// TIA Portal project "PID 2" (V17)

(* hardware
DEVICE "S7-1500/ET200MP station_1"  S7-1500 station
   slot 0: "Rail_0"  Rack  6ES7 590-1***0-0AA0
   slot 1: "PLC_1"  CPU 1512C-1 PN  6ES7 512-1CK00-0AB0  V2.1
      slot 3: "CPU display_1"  6ES7591-1AA00-0AA0
      slot 32768: "PROFINET interface_1"  X1
         slot 32769: "Port_1"  X1 P1
         slot 32770: "Port_2"  X1 P2
*)

// ===== PLC "PLC_1"  CPU 1512C-1 PN =====

VAR_GLOBAL   // PLC tag table "Default tag table"
   "System_Byte" AT %MB300 : Byte;
   "FirstScan" AT %M300.0 : Bool;
   "DiagStatusUpdate" AT %M300.1 : Bool;
   "AlwaysTRUE" AT %M300.2 : Bool;
   "AlwaysFALSE" AT %M300.3 : Bool;
   "Clock_Byte" AT %MB100 : Byte;
   "Clock_10Hz" AT %M100.0 : Bool;
   "Clock_5Hz" AT %M100.1 : Bool;
   "Clock_2.5Hz" AT %M100.2 : Bool;
   "Clock_2Hz" AT %M100.3 : Bool;
   "Clock_1.25Hz" AT %M100.4 : Bool;
   "Clock_1Hz" AT %M100.5 : Bool;
   "Clock_0.625Hz" AT %M100.6 : Bool;
   "Clock_0.5Hz" AT %M100.7 : Bool;
   "FRIO ANALÓGICA" AT %QD0 : Real;
   "CALOR ANALÓGICA" AT %QD4 : Real;
   "COMPUERTAS EXTERIOR" AT %Q8.0 : Bool;
   "COMPUERTA INTERIOR" AT %Q8.1 : Bool;
   "CALOR EXTERIOR ANALÓGICA" AT %QD10 : Real;
   "FRIO EXTERIOR ANALÓGICA" AT %QD14 : Real;
END_VAR

DATA_BLOCK "Data_block_1"   // DB2
{ S7_Optimized_Access := 'TRUE' }
VERSION : 0.1
   VAR
      "TEMPERATURA INTERIOR" : Real;
      "TEMPERATURA EXTERIOR" : Real;
      "FRIO INADECUADO" : Bool;
      "CALOR INADECUADO" : Bool;
      "FRIO EXTERIOR INADECUADO" : Bool;
      "CALOR EXTERIOR INADECUADO" : Bool;
   END_VAR
BEGIN
END_DATA_BLOCK

FUNCTION "FC_CONTROL PID" : Void   // FC1, LAD
{ S7_Optimized_Access := 'TRUE' }
VERSION : 0.1
BEGIN

REGION Network 1
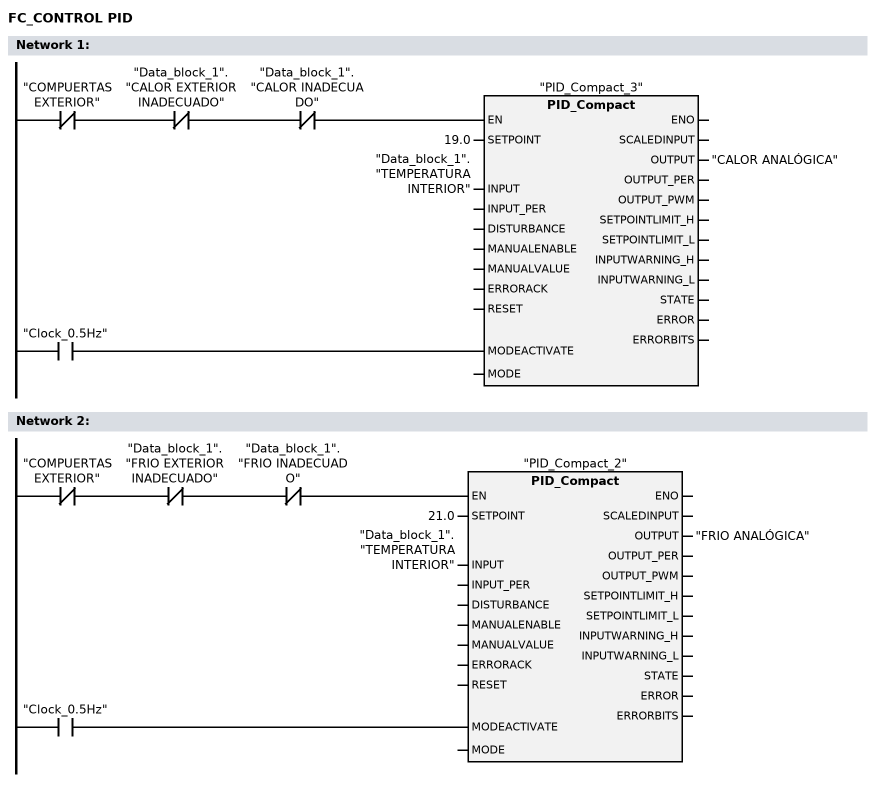
   IF NOT "COMPUERTAS EXTERIOR" AND NOT "Data_block_1"."CALOR EXTERIOR INADECUADO" AND NOT "Data_block_1"."CALOR INADECUADO" THEN
       "PID_Compact_3"(Setpoint := 19.0,   // PID_Compact
                       Input := "Data_block_1"."TEMPERATURA INTERIOR",
                       ModeActivate := "Clock_0.5Hz",
                       Output => "CALOR ANALÓGICA");
   END_IF;
END_REGION

REGION Network 2
   IF NOT "COMPUERTAS EXTERIOR" AND NOT "Data_block_1"."FRIO EXTERIOR INADECUADO" AND NOT "Data_block_1"."FRIO INADECUADO" THEN
       "PID_Compact_2"(Setpoint := 21.0,   // PID_Compact
                       Input := "Data_block_1"."TEMPERATURA INTERIOR",
                       ModeActivate := "Clock_0.5Hz",
                       Output => "FRIO ANALÓGICA");
   END_IF;
END_REGION
END_FUNCTION

FUNCTION "FC_MARCAS" : Void   // FC2, LAD
{ S7_Optimized_Access := 'TRUE' }
VERSION : 0.1
BEGIN

REGION Network 1
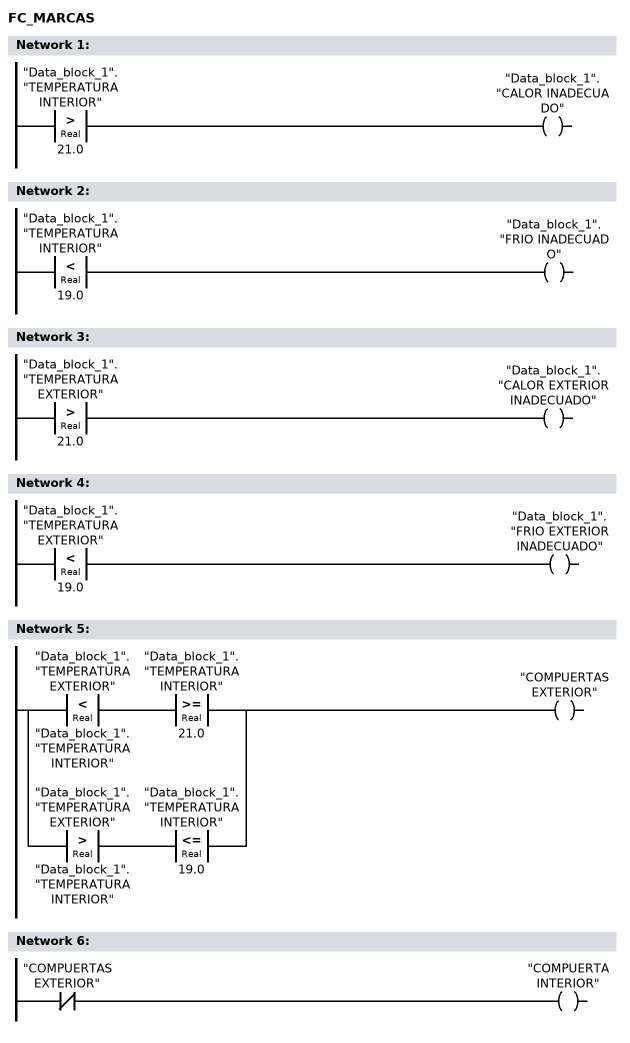
   RUNG wire#powerrail
      { S7_Templates := "SrcType := Real" } GT_Contact(in1 := "Data_block_1"."TEMPERATURA INTERIOR", in2 := 21.0)
      Coil( "Data_block_1"."CALOR INADECUADO" )
   END_RUNG
   // the same network as SCL:
   "Data_block_1"."CALOR INADECUADO" := "Data_block_1"."TEMPERATURA INTERIOR" > 21.0;
END_REGION

REGION Network 2
   RUNG wire#powerrail
      { S7_Templates := "SrcType := Real" } LT_Contact(in1 := "Data_block_1"."TEMPERATURA INTERIOR", in2 := 19.0)
      Coil( "Data_block_1"."FRIO INADECUADO" )
   END_RUNG
   // the same network as SCL:
   "Data_block_1"."FRIO INADECUADO" := "Data_block_1"."TEMPERATURA INTERIOR" < 19.0;
END_REGION

REGION Network 3
   RUNG wire#powerrail
      { S7_Templates := "SrcType := Real" } GT_Contact(in1 := "Data_block_1"."TEMPERATURA EXTERIOR", in2 := 21.0)
      Coil( "Data_block_1"."CALOR EXTERIOR INADECUADO" )
   END_RUNG
   // the same network as SCL:
   "Data_block_1"."CALOR EXTERIOR INADECUADO" := "Data_block_1"."TEMPERATURA EXTERIOR" > 21.0;
END_REGION

REGION Network 4
   RUNG wire#powerrail
      { S7_Templates := "SrcType := Real" } LT_Contact(in1 := "Data_block_1"."TEMPERATURA EXTERIOR", in2 := 19.0)
      Coil( "Data_block_1"."FRIO EXTERIOR INADECUADO" )
   END_RUNG
   // the same network as SCL:
   "Data_block_1"."FRIO EXTERIOR INADECUADO" := "Data_block_1"."TEMPERATURA EXTERIOR" < 19.0;
END_REGION

REGION Network 5
   RUNG wire#powerrail
      { S7_Templates := "SrcType := Real" } LT_Contact(in1 := "Data_block_1"."TEMPERATURA EXTERIOR", in2 := "Data_block_1"."TEMPERATURA INTERIOR")
      { S7_Templates := "SrcType := Real" } GE_Contact(in1 := "Data_block_1"."TEMPERATURA INTERIOR", in2 := 21.0)
      wire#w1
      Coil( "COMPUERTAS EXTERIOR" )
   END_RUNG
   RUNG wire#powerrail
      { S7_Templates := "SrcType := Real" } GT_Contact(in1 := "Data_block_1"."TEMPERATURA EXTERIOR", in2 := "Data_block_1"."TEMPERATURA INTERIOR")
      { S7_Templates := "SrcType := Real" } LE_Contact(in1 := "Data_block_1"."TEMPERATURA INTERIOR", in2 := 19.0)
   END_RUNG wire#w1
   // the same network as SCL:
   "COMPUERTAS EXTERIOR" := (("Data_block_1"."TEMPERATURA EXTERIOR" < "Data_block_1"."TEMPERATURA INTERIOR") AND ("Data_block_1"."TEMPERATURA INTERIOR" >= 21.0)) OR (("Data_block_1"."TEMPERATURA EXTERIOR" > "Data_block_1"."TEMPERATURA INTERIOR") AND ("Data_block_1"."TEMPERATURA INTERIOR" <= 19.0));
END_REGION

REGION Network 6
   RUNG wire#powerrail
      I_Contact( "COMPUERTAS EXTERIOR" )
      Coil( "COMPUERTA INTERIOR" )
   END_RUNG
   // the same network as SCL:
   "COMPUERTA INTERIOR" := NOT "COMPUERTAS EXTERIOR";
END_REGION
END_FUNCTION

ORGANIZATION_BLOCK "Main"   // OB1, LAD, ProgramCycle
TITLE = "Main Program Sweep (Cycle)"
{ S7_Optimized_Access := 'TRUE' }
VERSION : 0.1
   VAR_INPUT
      Initial_Call : Bool;   // Initial call of this OB
      Remanence : Bool;   // =True, if remanent data are available
   END_VAR
BEGIN

REGION Network 1
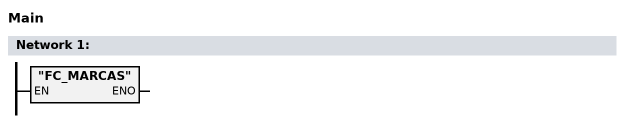
   RUNG wire#powerrail
      "FC_MARCAS"()
   END_RUNG
   // the same network as SCL:
   "FC_MARCAS"();
END_REGION
END_ORGANIZATION_BLOCK

ORGANIZATION_BLOCK "Cyclic interrupt"   // OB30, LAD, CyclicInterrupt
{ S7_Optimized_Access := 'TRUE' }
VERSION : 0.1
   VAR_INPUT
      Initial_Call : Bool;   // Initial call of this OB
      Event_Count : Int;   // Events discarded
   END_VAR
BEGIN

REGION Network 1
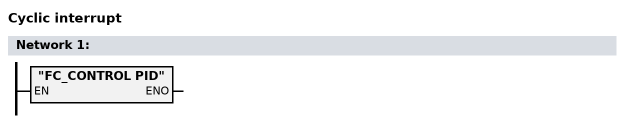
   RUNG wire#powerrail
      "FC_CONTROL PID"()
   END_RUNG
   // the same network as SCL:
   "FC_CONTROL PID"();
END_REGION
END_ORGANIZATION_BLOCK